FUNCTION_BLOCK VSG_ControlOfOutputs
VAR_INPUT
END_VAR
VAR_OUTPUT
END_VAR
VAR
END_VAR

// NETWORK 1

END_FUNCTION_BLOCK

(* stored: Version 1.1.0.1, ProductVersion 3.1.4024.15
   POU VSG_ControlOfOutputs: Id {cc759666-2ef0-42db-8b8f-79d5146704c2}, SpecialFunc None *)
